TYPE ST_MESSAGE_STATE :
STRUCT
  State         : E_MESSAGE_STATE;  // as always... combined value of Cmd equivalent and e_progress
END_STRUCT
END_TYPE

(* stored: Version 1.1.0.1, ProductVersion 3.1.4026.13
   DUT ST_MESSAGE_STATE: Id {9e66822f-d351-457c-b6e2-8ff98dc4e696} *)
